TYPE PositioningControl :
STRUCT
	Execute : BOOL;
	EmergencyStop : BOOL;
END_STRUCT
END_TYPE

(* stored: Version 1.1.0.1, ProductVersion 3.1.4024.9
   DUT PositioningControl: Id {ed08eca5-b9f3-423a-a3bd-c3a139899b46} *)
